(* Schneider Machine Expert - Basic project Project1_Part1CX, file version 1.6.0.0 *)
(* ProjectInformations: Name=New project *)

HARDWARE
  Cpu 0: TM221M16R/G
  EthernetConfiguration: NetworkName=M221, IpAllocationMode=FixedAddress, IpAddress=0.0.0.0, SubnetMask=0.0.0.0
  SerialLineConfiguration: Baud=Baud19200, Parity=ParityEven, DataBits=DataBits8, StopBits=StopBits1, PhysicalMedium=PhysicalMediumRs485, TransmissionMode=TransmissionModeModbusRtu, SlaveId=1, Addressing=SlaveAddressing
  MastTask: UsePeriodScanMode=false, PeriodScan=100
  FastTask: Period=255
  CpuBehavior: StartingMode=StartAsPreviousState, AutoSaveRamOnEeprom=true, WatchdogPeriod=250

SYMBOLS  (address, symbol, comment, settings)
  %TM0        [Type=TP, Preset=5, Base=OneSecond]
  %C1         "Count down from 5"  [Preset=5]
  %IW0.0      [Type=Type_0_10V, Scope=Scope_Normal, Minimum=0, Maximum=1000]
  %IW0.1      [Type=Type_0_10V, Scope=Scope_Normal, Minimum=0, Maximum=1000]

POU Project1-Part1B
  (* SectionNumber=1 *)

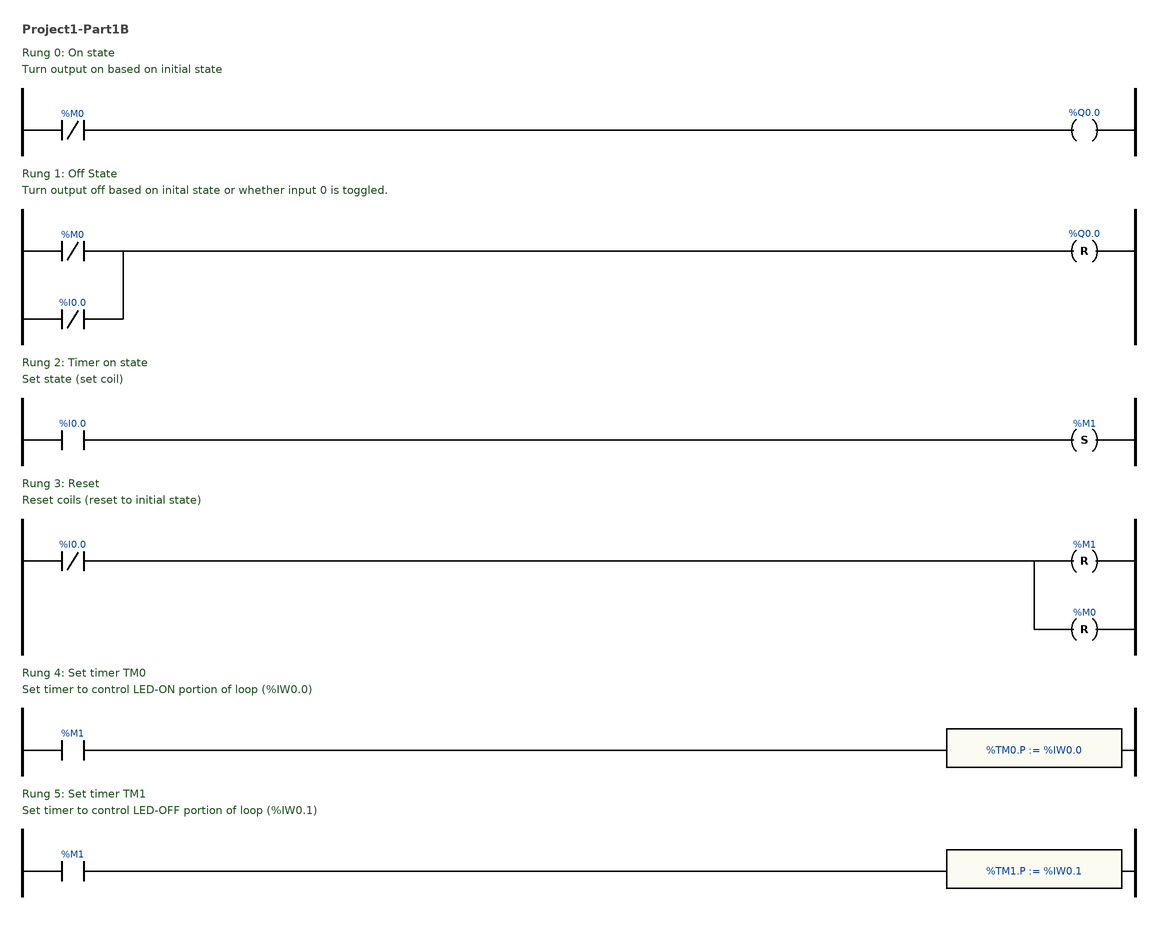

// Rung 0: On state
// Turn output on based on initial state
  LDN %M0
  ST %Q0.0
  // as ST:
  //   %Q0.0 := NOT %M0;

// Rung 1: Off State
// Turn output off based on inital state or whether input 0 is toggled.
  LDN %M0
  ORN %I0.0
  R %Q0.0
  // as ST:
  //   IF NOT %M0 OR NOT %I0.0 THEN %Q0.0 := FALSE; END_IF;

// Rung 2: Timer on state
// Set state (set coil)
  LD %I0.0
  S %M1
  // as ST:
  //   IF %I0.0 THEN %M1 := TRUE; END_IF;

// Rung 3: Reset
// Reset coils (reset to initial state)
  LDN %I0.0
  R %M1
  R %M0
  // as ST:
  //   IF NOT %I0.0 THEN %M1 := FALSE; END_IF;
  //   IF NOT %I0.0 THEN %M0 := FALSE; END_IF;

// Rung 4: Set timer TM0
// Set timer to control LED-ON portion of loop (%IW0.0)
  LD %M1
  [ %TM0.P := %IW0.0 ]
  // as ST:
  //   IF %M1 THEN %TM0.P := %IW0.0; END_IF;

// Rung 5: Set timer TM1
// Set timer to control LED-OFF portion of loop (%IW0.1)
  LD %M1
  [ %TM1.P := %IW0.1 ]
  // as ST:
  //   IF %M1 THEN %TM1.P := %IW0.1; END_IF;
